      L     "MAL1S021Par".Ilo.ILOMode;
      L     10;
      <>I   ;
      SPB   I10;
// man on
      U     "MAL1S021Par".Ilo.GrCMDManOn[1];
      S     "G009G".Gr.InManual; // GENERAL ELEMENTS GERM 5
      S     "G185M".Gr.InManual; // Traveling  Drive Germatingbox 5
      S     "G189M".Gr.InManual; // Turning Screws Germinationbox 5
      S     "G184M".Gr.InManual; // Wall locking Germatingbox 5
      S     "G182M".Gr.InManual; // Backwall moving Germatingbox 5
      S     "G183M".Gr.InManual; // Discharger locking Germatingbox 5
      R     "MAL1S021Par".Ilo.GrCMDManOn[1];
// man off
      U     "MAL1S021Par".Ilo.GrCMDManOff[1];
      S     "G009G".Gr.CmdManualOff; // GENERAL ELEMENTS GERM 5
      R     "G009G".Gr.InManual; // GENERAL ELEMENTS GERM 5
      S     "G185M".Gr.CmdManualOff; // Traveling  Drive Germatingbox 5
      R     "G185M".Gr.InManual; // Traveling  Drive Germatingbox 5
      R     "G185M".USW14; // ILO-cmd
      R     "G185M".USW15; // ILO-cmd
      S     "G189M".Gr.CmdManualOff; // Turning Screws Germinationbox 5
      R     "G189M".Gr.InManual; // Turning Screws Germinationbox 5
      R     "G189M".USW14; // ILO-cmd
      R     "G189M".USW15; // ILO-cmd
      S     "G184M".Gr.CmdManualOff; // Wall locking Germatingbox 5
      R     "G184M".Gr.InManual; // Wall locking Germatingbox 5
      S     "G183M".Gr.CmdManualOff; // Discharger locking Germatingbox 5
      R     "G183M".Gr.InManual; // Discharger locking Germatingbox 5
      S     "G182M".Gr.CmdManualOff; // Backwall moving Germatingbox 5
      R     "G182M".Gr.InManual; // Backwall moving Germatingbox 5
      R     "MAL1S021Par".Ilo.GrCMDManOff[1];
      R     "MAL1S021Par".Ilo.GrCMDManAdditional.Cmd1[1];
      R     "MAL1S021Par".Ilo.GrCMDManAdditional.Cmd2[1];
// man start
      U     "G187M".A_2511_KCL01I1.InpTrue; // pushbutton "start screws"
      S     "G009G".Gr.CmdOn; // GENERAL ELEMENTS GERM 5
      S     "G009G".Gr.CmdContinue; // GENERAL ELEMENTS GERM 5
      S     "G189M".Gr.CmdOn; // Turning Screws Germinationbox 5
      S     "G189M".Gr.CmdContinue; // Turning Screws Germinationbox 5
      S     "G185M".Gr.CmdOn; // Traveling  Drive Germatingbox 5
      S     "G185M".Gr.CmdContinue; // Traveling  Drive Germatingbox 5
      U     "MAL1S021Par".Ilo.GrCMDManStart[1];
      R     "MAL1S021Par".Ilo.GrCMDManStart[1];
      U     "MAL1S021Par".Ilo.GrCMDManStart[2];
      R     "MAL1S021Par".Ilo.GrCMDManStart[2];
// man stop
      UN    "G187M".A_2511_KCL01I2.InpTrue; // pushbutton "stop screws"  //dyk 081025 Inverted
      S     "G189M".Gr.CmdOff; // Turning Screws Germinationbox 5
      U     "MAL1S021Par".Ilo.GrCMDManStop[1];
      O(    ;
      UN    "G187M".A_2511_KCL01I3.InpTrue; // pushbutton "drive fwd"
      UN    "G187M".A_2511_KCL01I4.InpTrue; // pushbutton "drive rev"
      )     ;
      S     "G185M".Gr.CmdOff; // Traveling  Drive Germatingbox 5

      UN    "G184M".Gr.InManual; // Wall locking Germatingbox 5
      O(    ;
      UN    "G187M".A_2515_KCL01I5.InpTrue; // pushbutton "locking"
      UN    "G187M".A_2515_KCL01I6.InpTrue; // pushbutton "unlocking"
      )     ;
      S     "G184M".Gr.CmdOff; // Wall locking/unlocking Germatingbox 5

      UN    "G183M".Gr.InManual; // discharger coupling Germatingbox 5
      O(    ;
      UN    "G187M".A_2515_KCL01I4.InpTrue; // pushbutton "discharger coupling"
      UN    "G187M".A_2515_KCL01I3.InpTrue; // pushbutton "discharger uncoupling"
      )     ;
      S     "G183M".Gr.CmdOff; // discharger coupling Germatingbox 5

      UN    "G182M".Gr.InManual; // Backwall moving Germatingbox 5
      O(    ;
      UN    "G187M".A_2515_KCL01I1.InpTrue; // pushbutton "backwall lifting"
      UN    "G187M".A_2515_KCL01I2.InpTrue; // pushbutton "backwall lowerring"
      )     ;
      S     "G182M".Gr.CmdOff; // Backwall moving Germatingbox 5

      U     "MAL1S021Par".Ilo.GrCMDManStop[1];
      R     "MAL1S021Par".Ilo.GrCMDManStop[1];
// man fault reset
      U     "MAL1S021Par".Ilo.GrCMDManFaultReset[1];
      S     "G009G".Gr.CmdFaultReset; // GENERAL ELEMENTS GERM 5
      S     "G185M".Gr.CmdFaultReset; // Traveling  Drive Germatingbox 5
      S     "G189M".Gr.CmdFaultReset; // Turning Screws Germinationbox 5
      R     "MAL1S021Par".Ilo.GrCMDManFaultReset[1];
      NOP   0;
// Manual wall locking
      UN    "G184M".Gr.InManual; // Wall locking Germatingbox 5
      ON    "G187M".A_2515_KCL01I5.InpTrue; // pushbutton "locking"
      SPB   f102;
      S     "G184M".Gr.CmdOn; // Wall locking/unlocking Germatingbox 5
f102: NOP   0;
// Manual wall unlocking
      UN    "G184M".Gr.InManual; // Wall locking Germatingbox 5
      ON    "G187M".A_2515_KCL01I6.InpTrue; // pushbutton "unlocking"
      SPB   f103;
      S     "G184M".Gr.CmdOn; // Wall locking/unlocking Germatingbox 5
f103: NOP   0;
// Manual discharger coupling
      UN    "G183M".Gr.InManual; // discharger coupling Germatingbox 5
      ON    "G187M".A_2515_KCL01I4.InpTrue; // pushbutton "discharger coupling"
      SPB   f104;
      S     "G183M".Gr.CmdOn; // discharger coupling Germatingbox 5
f104: NOP   0;
// Manual discharger uncoupling
      UN    "G183M".Gr.InManual; // discharger coupling Germatingbox 5
      ON    "G187M".A_2515_KCL01I3.InpTrue; // pushbutton "discharger uncoupling"
      SPB   f105;
      S     "G183M".Gr.CmdOn; // discharger coupling Germatingbox 5
f105: NOP   0;
// Manual backwall moving
      UN    "G182M".Gr.InManual; // Backwall moving Germatingbox 5
      ON    "G187M".A_2515_KCL01I1.InpTrue; // pushbutton "backwall lifting"
      SPB   f106;
      S     "G182M".Gr.CmdOn; // Backwall moving Germatingbox 5
f106: NOP   0;
      UN    "G182M".Gr.InManual; // Backwall moving Germatingbox 5
      ON    "G187M".A_2515_KCL01I2.InpTrue; // pushbutton "backwall lowerring"
      SPB   f107;
      S     "G182M".Gr.CmdOn; // Backwall moving Germatingbox 5
f107: NOP   0;
// manual direction
      UN    "G185M".Gr.InManual; // Traveling  Drive Germatingbox 5
      O     ;
      UN    "G187M".A_2511_KCL01I3.InpTrue; // pushbutton "drive fwd"
      UN    "G187M".A_2511_KCL01I4.InpTrue; // pushbutton "drive rev"
      SPB   f109;
      U     "G187M".A_2511_KCL01I3.InpTrue; // pushbutton "drive fwd"
      =     "G185M".USW14; // ILO-cmd run fwd
      S     "G185M".Gr.CmdOn; // Traveling  Drive Germatingbox 5
      U     "G187M".A_2511_KCL01I4.InpTrue; // pushbutton "drive rev"
      =     "G185M".USW15; // ILO-cmd run rev
      S     "G185M".Gr.CmdOn; // Traveling  Drive Germatingbox 5

// target position
      L     "MAL1S021Par".Ilo.SetpointInt01[1];
      T     "MAL1S021Par".Par.ParIntProcess.Speed_ILO_FloorRotating;
f109: NOP   0;

I10:  NOP   0;
//
// copy state
      U     "G185M".Gr.InOutAutostartMan; // TRAVELLING DRIVE  GERM 5
      =     "MAL1S021Par".Ilo.GrSTMan[2];
      U     "G189M".Gr.InOutAutostartMan; // TURNING SCREWS  GERM 5
      =     "MAL1S021Par".Ilo.GrSTMan[6];
      U     "G190M".Gr.InOutAutostartMan; // FAN AND VALVE SRAY AIR  GERM 5
      =     "MAL1S021Par".Ilo.GrSTMan[7];
      U     "G191M".Gr.InOutAutostartMan; // FRESH AIR LOUVER  GERM 5
      =     "MAL1S021Par".Ilo.GrSTMan[8];
      U     "G197M".Gr.InOutAutostartMan; // COOLING / HEATING  GERM 5
      =     "MAL1S021Par".Ilo.GrSTMan[14];

// copy state

NETWORK
TITLE =ASW_9999: Init ASW Flags
// clear all flags explicde to find them back
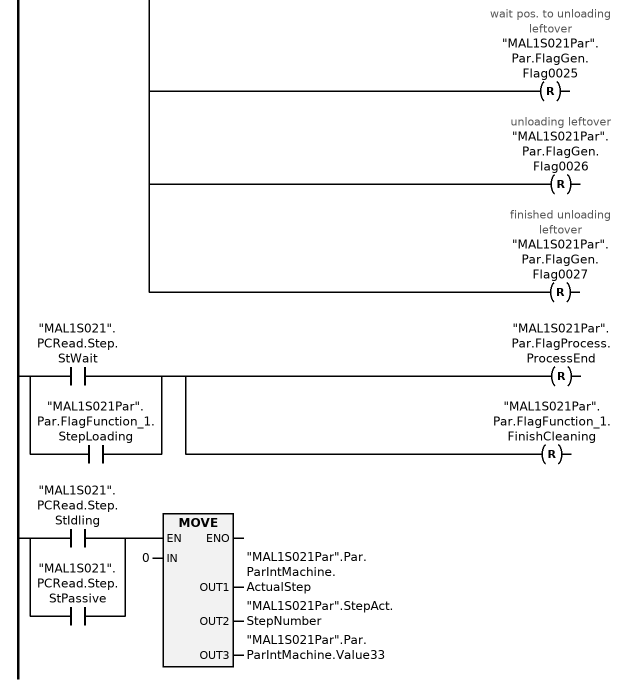
      U     "MAL1S021".PCRead.Step.StIdling;
      O     "MAL1S021".PCRead.Step.StPassive;
      R     "MAL1S021Par".Par.FlagFunction_1.StepLoading;
      R     "MAL1S021Par".Par.FlagFunction_1.StepUnloading;
      R     "MAL1S021Par".Par.FlagFunction_1.StepCleaning;
      R     "MAL1S021Par".Par.FlagFunction_1.LoadingBreak;
      R     "MAL1S021Par".Par.FlagFunction_1.UnloadingBreak;
      R     "MAL1S021Par".Par.FlagFunction_1.CleaningBreak;
      R     "MAL1S021Par".Par.FlagFunction_1.FinishLoading;
      R     "MAL1S021Par".Par.FlagFunction_1.FinishUnloading;
      R     "MAL1S021Par".Par.FlagFunction_1.FinishCleaning;
      R     "MAL1S021Par".Par.FlagFunction_1.Round_1;
      R     "MAL1S021Par".Par.FlagFunction_1.Round_2;
      R     "MAL1S021Par".Par.FlagFunction_1.Round_3;
      R     "MAL1S021Par".Par.FlagFunction_1.Round_4;
      R     "MAL1S021Par".Par.FlagFunction_1.Round_5;
      R     "MAL1S021Par".Par.FlagFunction_1.Round_6;
      R     "MAL1S021Par".Par.FlagFunction_1.Beladung_beendet;
      R     "MAL1S021Par".Par.FlagFunction_1.Entladerunden_erreicht;
      R     "MAL1S021Par".Par.FlagFunction_1.Reinigungsrunde_erreicht;
      R     "MAL1S021Par".Par.FlagGen.TurningStarted;
      R     "MAL1S021Par".Par.FlagFunction_1.TurningStart;
      R     "MAL1S021Par".Par.FlagFunction_1.TurningStop;
      R     "MAL1S021Par".Par.FlagFunction_1.TurningLeft;
      R     "MAL1S021Par".Par.FlagFunction_1.TurningRight;
      R     "MAL1S021Par".Par.FlagFunction_1.LoadFirstPartEnd;
      R     "MAL1S021Par".Par.FlagFunction_1.TurningWithSpraying;
      R     "MAL1S021Par".Par.FlagFunction_1.TurningWithoutSpraying;
      R     "MAL1S021Par".Par.FlagGen.TurningStarted;
      R     "MAL1S021Par".Par.FlagProcess2.Turning1WithoutSpraying;
      R     "MAL1S021Par".Par.FlagProcess2.Turning2WithoutSpraying;
      R     "MAL1S021Par".Par.FlagProcess2.Turning1WithSpraying;
      R     "MAL1S021Par".Par.FlagProcess2.Turning2WithSpraying;
      R     "MAL1S021Par".Par.FlagProcess2.Turning1WithDosing;
      R     "MAL1S021Par".Par.FlagProcess2.Turning2WithDosing;
      R     "MAL1S021Par".Par.FlagProcess2.StartFirstTurningRound;
      R     "MAL1S021Par".Par.FlagProcess2.StartSecondTurningRound;

      R     "MAL1S021Par".Par.FlagFunction_1.UnloadFirstPartEnd;
      R     "MAL1S021Par".Par.FlagFunction_1.UnloadSecondPartEnd;
      R     "MAL1S021Par".Par.FlagFunction_1.UnloadFirstPart;
      R     "MAL1S021Par".Par.FlagFunction_1.UnloadSecondPart;
      R     "MAL1S021Par".Par.FlagFunction_1.UnloadingStarted;
      R     "MAL1S021Par".Par.FlagProcess.ProcessActive;
      R     "MAL1S021Par".Par.FlagProcess.ProcessStartFP;
      R     "MAL1S021Par".Par.FlagProcess.ProcessStartScan;
      R     "MAL1S021Par".Par.FlagProcess.ProcessEnd;
      R     "MAL1S021Par".Par.FlagProcess.FP_SendResultToPIC;
      R     "MAL1S021Par".Par.FlagMachine.ImpulsNullstellung;
      R     "MAL1S021Par".Par.FlagMachine_0.CmdTurnRevAfterUnloading;
      R     "MAL1S021Par".Par.FlagMachine_0.CleaningAfterUnloading;
      R     "MAL1S021Par".Par.FlagMachine_0.CleaningAfterLoading;

      R     "MAL1S021Par".Par.FlagGen.Flag0024; // finished first unloading
      R     "MAL1S021Par".Par.FlagGen.Flag0025; // wait pos. to unloading leftover
      R     "MAL1S021Par".Par.FlagGen.Flag0026; // unloading leftover
      R     "MAL1S021Par".Par.FlagGen.Flag0027; // finished unloading leftover

//
      U     "MAL1S021".PCRead.Step.StWait;
      O     "MAL1S021Par".Par.FlagFunction_1.StepLoading;
      R     "MAL1S021Par".Par.FlagProcess.ProcessEnd;
      R     "MAL1S021Par".Par.FlagFunction_1.FinishCleaning;

      U     "MAL1S021".PCRead.Step.StIdling;
      O     "MAL1S021".PCRead.Step.StPassive;
      SPBN  csn;
      L     0; // clear step number
      T     "MAL1S021Par".Par.ParIntMachine.ActualStep;
      T     "MAL1S021Par".StepAct.StepNumber;
      T     "MAL1S021Par".Par.ParIntMachine.Value33; //aktuelle Wartezeit Maschine bei 100% Unloading-Position
csn:  NOP   0;

NETWORK
TITLE =Main0_End: Init flag
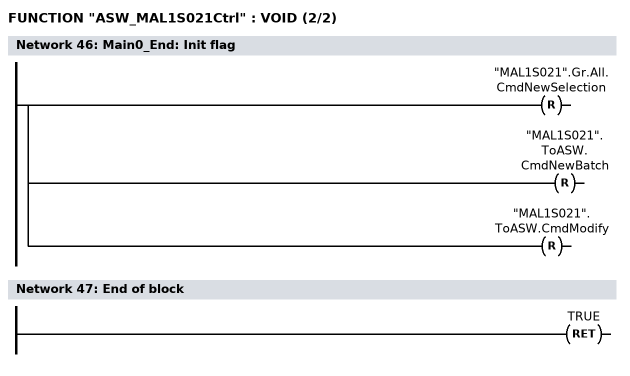

      SET   ;
      R     "MAL1S021".Gr.All.CmdNewSelection;
      R     "MAL1S021".ToASW.CmdNewBatch;
      R     "MAL1S021".ToASW.CmdModify;

NETWORK
TITLE =End of block

      BE    ;

END_FUNCTION

